FUNCTION_BLOCK FB_LamparaConmutada_LD
VAR_INPUT
END_VAR
VAR_OUTPUT
END_VAR
VAR
    Pulsacion: R_TRIG;
    
    Lampara AT %Q*: BOOL;
    Pulsador AT %I*: BOOL;    
END_VAR

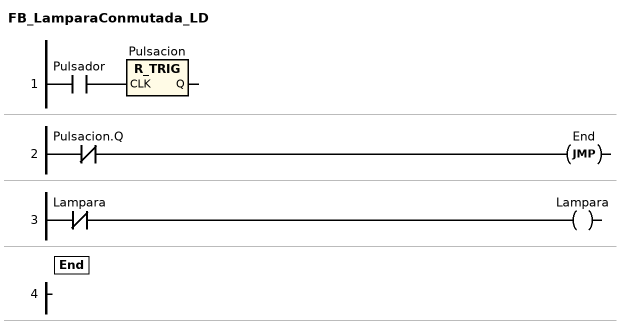
// NETWORK 1
Pulsacion(CLK := Pulsador); // R_TRIG

// NETWORK 2
IF NOT Pulsacion.Q THEN JMP End; END_IF

// NETWORK 3
Lampara := NOT Lampara;

// NETWORK 4
End: ;

END_FUNCTION_BLOCK

(* stored: Version 1.1.0.1, ProductVersion 3.1.4024.15
   POU FB_LamparaConmutada_LD: Id {fb9e8f1e-35ac-4616-995f-8d9dee686820}, SpecialFunc None *)
